// Brief: Setup Arm Self-check
FUNCTION_BLOCK PUBLIC FB_SetupCtrlSelfCheck EXTENDS FB_SetupArmCtrlBase
VAR_INPUT
END_VAR
VAR_OUTPUT
END_VAR
VAR

	
END_VAR

METHOD PUBLIC init : BOOL
VAR_IN_OUT CONSTANT
	i_setupArm	:FB_SetupArm;
END_VAR
VAR_IN_OUT 
	r_setupArmCtrlCmd :ST_SetupArmCtrlCmds;
END_VAR
SUPER^.Init(i_setupArm,r_setupArmCtrlCmd);
END_METHOD

END_FUNCTION_BLOCK

(* stored: Version 1.1.0.1, ProductVersion 3.1.4024.12
   POU FB_SetupCtrlSelfCheck: Id {de863df1-4a4d-4fa9-a2ab-b3b6dd7ec2a1}, SpecialFunc None
   Method init: Id {57d7becd-4a0a-4f37-8764-94cf78ff725a} *)
